FUNCTION_BLOCK FB_P_Control
VAR_INPUT
	ProcessVariable : LREAL;
	Setpoint 		: LREAL;
	Kp 				: LREAL;
END_VAR         	
VAR_OUTPUT      	
	Term 			: LREAL;
END_VAR

Term := (Setpoint - ProcessVariable) * Kp;

END_FUNCTION_BLOCK

(* stored: Version 1.1.0.1, ProductVersion 3.1.4022.3
   POU FB_P_Control: Id {5b99849f-1fb0-4200-b85f-0d13e85c0b7e}, SpecialFunc None *)
